// Mitsubishi GX Works2 project: 3번 반복   PLC: Q02/Q02H

PROGRAM MAIN
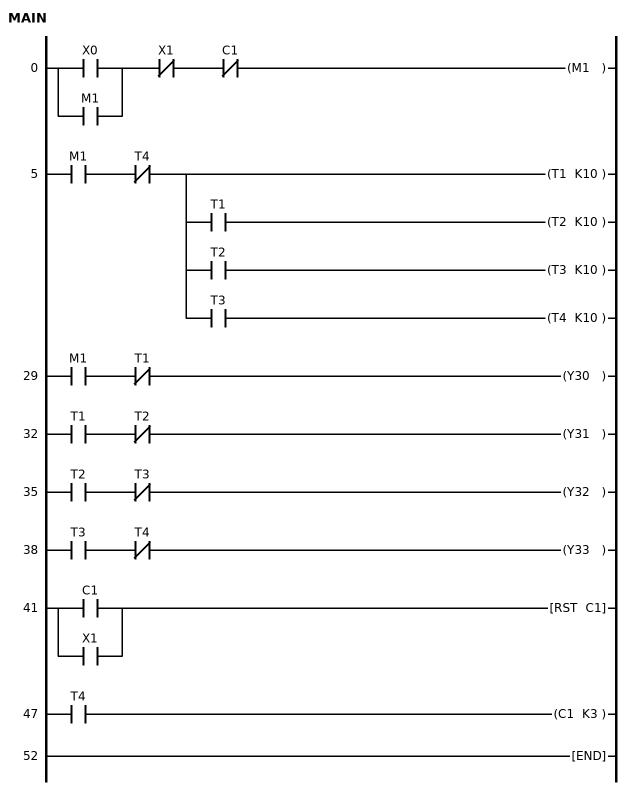
0     LD      X0
      OR      M1
      ANI     X1
      ANI     C1
      OUT     M1
5     LD      M1
      ANI     T4
      OUT     T1 K10
      MPS
      AND     T1
      OUT     T2 K10
      MRD
      AND     T2
      OUT     T3 K10
      MPP
      AND     T3
      OUT     T4 K10
29    LD      M1
      ANI     T1
      OUT     Y30
32    LD      T1
      ANI     T2
      OUT     Y31
35    LD      T2
      ANI     T3
      OUT     Y32
38    LD      T3
      ANI     T4
      OUT     Y33
41    LD      C1
      OR      X1
      RST     C1
47    LD      T4
      OUT     C1 K3
52    END
END_PROGRAM
